SUBAPPLICATION Uebung_215 (* Standard IEC 61131-3 FB_CTD (Rückwärtszähler, INT) mit Terminal-Ausgabe *)
  (* Standard: 61131-3; Description: Copyright (c) 2026 Meisterschulen am Ostbahnhof This program and the accompanying materials are made available under the terms of the Eclipse Public License 2.0 which is available at https://www.eclipse.org/legal/epl-2.0/ SPDX-License-Identifier: EPL-2.0 *)
  (* Version 1.1, 2026-04-21, Franz Höpfinger, Meisterschulen am Ostbahnhof, Added terminal output for counter value *)
  (* Version 1.0, 2026-04-20, Franz Höpfinger, Meisterschulen am Ostbahnhof, initial API and implementation (IEC 61131-3 version) *)
  PACKAGE Uebungen;
  IMPORT Uebungen::const::UT::DefaultPool::OutputNumber_N1;
  IMPORT logiBUS::io::DI::logiBUS_DI::Input_I1;
  IMPORT logiBUS::io::DI::logiBUS_DI::Input_I2;
  IMPORT logiBUS::io::DQ::logiBUS_DO::Output_Q1;
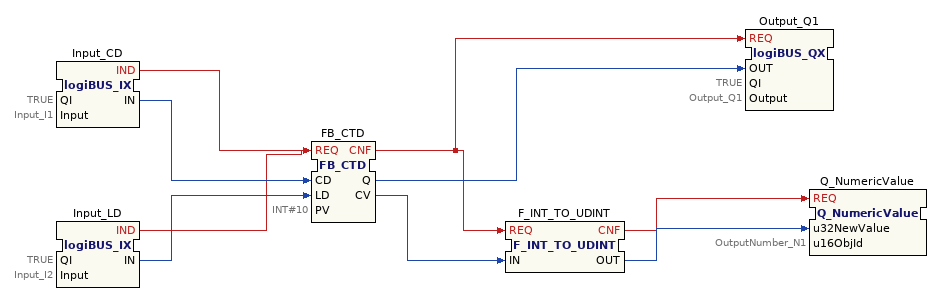
  (* F_INT_TO_UDINT ist großer Quatsch ... keine Negativen Zahlen möglich *)
  FBS
    FB_CTD : iec61131::counters::FB_CTD(PV := INT#10);
    Input_CD : logiBUS::io::DI::logiBUS_IX(QI := TRUE, Input := Input_I1);
    Input_LD : logiBUS::io::DI::logiBUS_IX(QI := TRUE, Input := Input_I2);
    Output_Q1 : logiBUS::io::DQ::logiBUS_QX(QI := TRUE, Output := Output_Q1);
    Q_NumericValue : isobus::UT::Q::Q_NumericValue(u16ObjId := OutputNumber_N1);
    F_INT_TO_UDINT : iec61131::conversion::F_INT_TO_UDINT;
  END_FBS
  EVENT_CONNECTIONS
    Input_CD.IND TO FB_CTD.REQ;
    Input_LD.IND TO FB_CTD.REQ;
    FB_CTD.CNF TO Output_Q1.REQ;
    FB_CTD.CNF TO F_INT_TO_UDINT.REQ;
    F_INT_TO_UDINT.CNF TO Q_NumericValue.REQ;
  END_CONNECTIONS
  DATA_CONNECTIONS
    Input_CD.IN TO FB_CTD.CD;
    Input_LD.IN TO FB_CTD.LD;
    FB_CTD.Q TO Output_Q1.OUT;
    FB_CTD.CV TO F_INT_TO_UDINT.IN;
    F_INT_TO_UDINT.OUT TO Q_NumericValue.u32NewValue;
  END_CONNECTIONS
END_SUBAPPLICATION
